FUNCTION Controleren_tijd : BOOL
VAR
  Huidige_tijd : INT; //Invoer van de tijd
END_VAR

IF (Huidige_tijd >= 0) AND (Huidige_tijd <= 2400) THEN
	IF Huidige_tijd >= 1000 THEN
		Controleren_tijd := TRUE
	ELSIF
		Controleren_tijd := FALSE
	END_IF
ELSE
	Controleren_tijd := FALSE //Geeft aan dat de ingevoerde tijd ongeldig is
END_IF;

END_FUNCTION

(* stored: Version 1.1.0.1, ProductVersion 3.1.4024.12
   POU Controleren_tijd: Id {16096a76-5c46-497a-8817-829de55f3d91}, SpecialFunc None *)
